TYPE ST_Area_Bedroom2 :
STRUCT
	wpRoom				: ST_WP_Bedroom2;
	fbSpotLights		: FB_DigitalOut;
END_STRUCT
END_TYPE

(* stored: Version 1.1.0.1, ProductVersion 3.1.4024.12
   DUT ST_Area_Bedroom2: Id {2008dc79-91ed-4b72-8f96-fbe5444c9e80} *)
